{attribute 'no_explicit_call' := 'Observable is a CLASS and must be accessed using methods or properties'}
FUNCTION_BLOCK Observable IMPLEMENTS I_Observable
VAR
	verbose							: BOOL := TRUE;
	// Make sure the list of references to subscribers is updated after online change 
	observers						: ARRAY[1..param.MaxObservers] OF I_Observer;
END_VAR


// The body of a class must not be used for code.  
// Cyclic code should be called from a method if needed.

METHOD Attach : BOOL
VAR_INPUT
	observer			: I_Observer;
END_VAR
VAR
	i					: INT;
END_VAR
(* default *)
attach := FALSE;

(* loop if the subscriber is already registered *)
FOR i := 1 TO param.MaxObservers DO
	IF observers[i] = observer 	THEN
		observer.update();
		attach := TRUE;
		RETURN;
	END_IF
END_FOR

(* loop for first free position if not yet attached *)
FOR i := 1 TO param.MaxObservers DO
	IF observers[i] = 0 	THEN
		observers[i] := observer;
		message('Observer registered');
		observer.update();
		attach := TRUE;
		EXIT;
	END_IF
END_FOR
END_METHOD

METHOD Detach : BOOL
VAR_INPUT
	observer			: I_Observer;
END_VAR
VAR
	i					: INT;
END_VAR
(* default *)
detach := FALSE;

(* loop if the subscriber is already registered *)
FOR i := 1 TO param.MaxObservers DO
	IF observers[i] = observer 	THEN
		observers[i] := 0;
		message('Observer deregistered');
		detach := TRUE;
		RETURN;
	END_IF
END_FOR
END_METHOD

{attribute 'call_after_online_change_slot' := '0'}
METHOD PRIVATE fbreinit
(*	!!!!!!!!!!!!!!!!!!!!!!!!!!!!!!!!!
   	THIS METHOD is force called after every online change 
   	!= the fb_reinit system call that will be called after the instance of the concerned function block has been copied 
 	(during an online change after modifications in the function block declaration)

	This is necessary since both observer en observee have references to one other
	!!!!!!!!!!!!!!!!!!!!!!!!!!!!!!!!!	*) 
VAR
	i					: INT;
END_VAR
(* loop if the subscriber is already registered *)
FOR i := 1 TO param.MaxObservers DO
	observers[i] := 0;
END_FOR
breinit:=NOT breinit; // flip the test marker
END_METHOD

METHOD PRIVATE Message : BOOL
VAR_INPUT
	strArg						: STRING;
END_VAR
// Log message
IF verbose  THEN
	ADSLOGSTR(
		msgCtrlMask := ADSLOG_MSGTYPE_HINT OR ADSLOG_MSGTYPE_LOG, // ADSLOG_MSGTYPE_ERROR OR ADSLOG_MSGTYPE_LOG, 
		msgFmtStr 	:= '%s',
		strArg 		:= strArg
		);
END_IF
END_METHOD

PROPERTY NoOfAttachedObservers : int
GET
VAR
	i							: INT;
END_VAR
// In stead of using an internal counter that could fail
// run through the array of attached observers
(* loop for first free position if not yet attached *)
NoOfAttachedObservers := 0;
FOR i := 1 TO param.MaxObservers DO
	IF observers[i] <> 0 	THEN
		NoOfAttachedObservers := NoOfAttachedObservers + 1;
	END_IF
END_FOR
END_GET
END_PROPERTY

METHOD Notify : BOOL
VAR
	i			: INT;
END_VAR
(* default *)
notify := FALSE;

(* loop if the subscriber is already registered *)
FOR i := 1 TO param.MaxObservers DO
	IF observers[i] <> 0 	THEN
		observers[i].update();
	END_IF
END_FOR
END_METHOD

END_FUNCTION_BLOCK

(* stored: Version 1.1.0.1, ProductVersion 3.1.4024.11
   POU Observable: Id {e2a73847-3ae9-41c4-a05d-e034052bdb33}, SpecialFunc None
   Method Attach: Id {8777bfbf-0b24-4d4c-bfbb-b615baf81400}
   Method Detach: Id {e9b4dda7-c343-4f9f-a3ca-f5b9e6583823}
   Method fbreinit: Id {5eb48304-7ea0-4c0a-aa2b-8367a1a8f441}
   Method Message: Id {bdd75991-46b2-4d02-b68d-98ecf52da978}
   Property NoOfAttachedObservers: Id {5bbf002f-f9f1-4de2-9982-3bdcbd5a4adc}
   Get Get: Id {a014369f-9eb1-4618-82ee-295f2393511e}
   Method Notify: Id {066cc371-6893-4a9d-a670-ce206a879997} *)
